Omron Sysmac Studio project modbus (Sysmac Studio 1.23.0.14, StandardProject)

# Controller new_Controller_0: NX1P2-1040DT1 version 1.18
Task PrimaryTask (priority 4, period or condition 2000): Programa0

VAR_GLOBAL CONSTANT
    Mi_Modulo485 : _sOPTBOARD_ID := (SlotNo := 2, IPAdr := [5(16#0)]);
END_VAR
VAR_GLOBAL
    Mi_Puerto : _sDEVICE_PORT;
    valor : INT;
    Escritura_20hz_Variador1 AT %W0.0 : BOOL;  (* published *)
    Escritura_50hz_Variador1 AT %W0.1 : BOOL;
END_VAR
VAR_GLOBAL RETAIN
    lectura_real AT %D0 : REAL;  (* published *)
END_VAR
VAR_GLOBAL
    run_fw : BOOL;
    run_bw : BOOL;
    stop_variador : BOOL;
    lectura_variador1 AT %W0.4 : BOOL;
    escritura_adelante_variador AT %W0.05 : BOOL;
    escritura_atras_variador AT %W0.06 : BOOL;
    escritura_marcha_variador AT %W0.2 : BOOL;
    escritura_paro_variador AT %W0.3 : BOOL;
    escritura_aceleracion1_variador : BOOL;
    escritura_aceleracion2_variador : BOOL;
END_VAR

PROGRAM Programa0
VAR
    Escritura_Frecuencia_Variador1 : BOOL;
    Instancia_Escritura_Frecuencia_Variador1 : NX_ModbusRtuWrite;
    Numero_Nodo_Variador1 : UINT;
    Trama_Escritura_Frecuencia_Variador1 : _sSERIAL_MODBUSRTU_WRITE;
    Datos_Escritura_Frecuencia_Variador1 : ARRAY[0..1] OF WORD;
    Option_Escritura_Frecuencia_Variador1 : _sSERIAL_MODBUSRTU_OPTION;
    Abort_Escritura_Frecuencia_Variador1 : BOOL;
    Busy_Escritura_Frecuencia_Variador1 : BOOL;
    CommandAborted_Escritura_Frecuencia_Variador1 : BOOL;
    Error_Escritura_Frecuencia_Variador1 : BOOL;
    ErrorID_Escritura_Frecuencia_Variador1 : BOOL;
    ErrorIDEX_Escritura_Frecuencia_Variador1 : BOOL;
    Instancia_Lectura_Frecuencia_Variador1 : NX_ModbusRtuRead;
    Trama_Lectura_Frecuencia_Variador1 : _sSERIAL_MODBUSRTU_READ;
    Datos_Lectura_Frecuencia_Variador1 : ARRAY[0..1] OF WORD;
    Option_Lectura_Frecuencia_Variador1 : _sSERIAL_MODBUSRTU_OPTION;
    Busy_Lectura_Frecuencia_Variador1 : BOOL;
    CommandAborted_Lectura_Frecuencia_Variador1 : BOOL;
    Error_Lectura_Frecuencia_Variador1 : BOOL;
    ErrorID_Lectura_Frecuencia_Variador1 : WORD;
    ErrorIDEX_Lectura_Frecuencia_Variador1 : DWORD;
    ReadSize_Lectura_Frecuencia_Variador1 : UINT;
    Abort_Lectura_Frecuencia_Variador1 : BOOL;
    nu : UINT;
    error : WORD;
    carmen : BOOL;
    pilo : BOOL;
    lectur : BOOL;
    Trama_Escritura_Marcha_Variador1 : _sSERIAL_MODBUSRTU_WRITE;
    Datos_Escritura_Marcha_Variador1 : BOOL;
    Option_Escritura_Marcha_Variador1 : _sSERIAL_MODBUSRTU_OPTION;
    Abort_Escritura_Marcha_Variador1 : BOOL;
    Trama_Escritura_Paro_Variador1 : _sSERIAL_MODBUSRTU_WRITE;
    Trama_Escritura_Sentido_Variador1 : _sSERIAL_MODBUSRTU_WRITE;
    Datos_Escritura_Sentido_Variador1 : BOOL;
    Option_Escritura_Sentido_Variador1 : _sSERIAL_MODBUSRTU_OPTION;
    Instancia_Escritura_Sentido_Variador1 : NX_ModbusRtuWrite;
    Datos_Escritura_Paro_Variador1 : BOOL;
    lectura_int : INT;
    Abort_Escritura_Sentido_Variador1 : BOOL;
    Trama_Escritura_Tiempo_Variador1 : _sSERIAL_MODBUSRTU_WRITE;
    Datos_Escritura_Tiempo_Variador1 : ARRAY[0..1] OF WORD;
    Option_Escritura_Tiempo_Variador1 : _sSERIAL_MODBUSRTU_OPTION;
    Abort_Escritura_Tiempo_Variador1 : BOOL;
END_VAR
VAR_EXTERNAL
    Mi_Puerto : _sDEVICE_PORT;
END_VAR
VAR_EXTERNAL CONSTANT
    Mi_Modulo485 : _sOPTBOARD_ID;
END_VAR
VAR_EXTERNAL
    Escritura_20hz_Variador1 : BOOL;
    Escritura_50hz_Variador1 : BOOL;
    lectura_variador1 : BOOL;
    escritura_adelante_variador : BOOL;
    escritura_atras_variador : BOOL;
    escritura_marcha_variador : BOOL;
    escritura_paro_variador : BOOL;
    lectura_real : REAL;
    escritura_aceleracion1_variador : BOOL;
    escritura_aceleracion2_variador : BOOL;
END_VAR

(* Section Escritura_Frecuencia_Variador1: ladder, written here as Structured Text *)

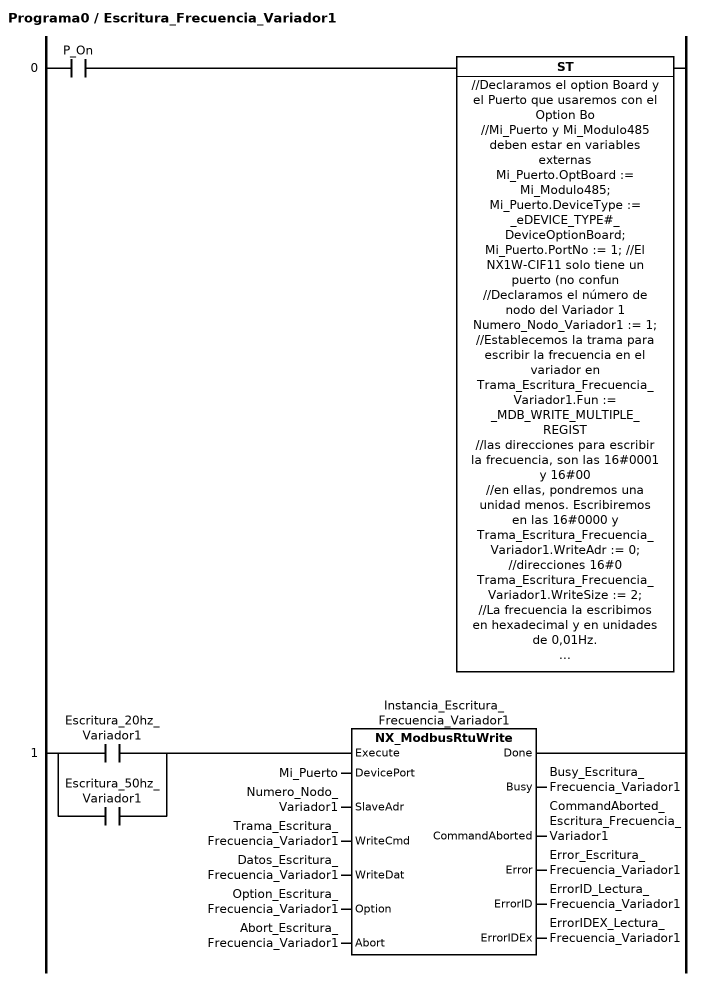
(* Rung 0 *)
IF P_On THEN
    //Declaramos el option Board y el Puerto que usaremos con el Option Board anterior.
    //Mi_Puerto y Mi_Modulo485 deben estar en variables externas
    Mi_Puerto.OptBoard := Mi_Modulo485;
    Mi_Puerto.DeviceType := _eDEVICE_TYPE#_DeviceOptionBoard;
    Mi_Puerto.PortNo := 1; //El NX1W-CIF11 solo tiene un puerto (no confundir con el slot donde está el módulo)
    
    //Declaramos el número de nodo del Variador 1
    Numero_Nodo_Variador1 := 1;
    
    //Establecemos la trama para escribir la frecuencia en el variador en los registros 0001h y 0002h
    Trama_Escritura_Frecuencia_Variador1.Fun := _MDB_WRITE_MULTIPLE_REGISTERS;
    //las direcciones para escribir la frecuencia, son las 16#0001 y 16#0002 pero como vamos a escribir
    //en ellas, pondremos una unidad menos. Escribiremos en las 16#0000 y 16#0001
    Trama_Escritura_Frecuencia_Variador1.WriteAdr := 0; //direcciones 16#0000 y 16#0001 para escribir la frecuencia
    Trama_Escritura_Frecuencia_Variador1.WriteSize := 2;
    
    //La frecuencia la escribimos en hexadecimal y en unidades de 0,01Hz. 5000 equivale a 50Hz.
    Datos_Escritura_Frecuencia_Variador1[0] := 0;
    IF Escritura_50hz_Variador1 THEN
    	Datos_Escritura_Frecuencia_Variador1[1] := 16#1388; //5000 en decimal que son 16#1388 (50Hz)
    ELSIF Escritura_20hz_Variador1 THEN
    	Datos_Escritura_Frecuencia_Variador1[1] := 16#07D0;
    END_IF;
    
    //establecemos que el TimeOut sea de 2 segundos (unidades de 0,1s) es el tiempo de espera
    //antes de dar por pérdida la comunicación y marcar el error 0400
    Option_Escritura_Frecuencia_Variador1.TimeOut := 20;
    
    //Activamos la comunicación poniendo la entrada Abort a False
    Abort_Escritura_Frecuencia_Variador1 := FALSE;
END_IF;
(* Rung 1 *)
Instancia_Escritura_Frecuencia_Variador1(Execute := Escritura_20hz_Variador1 OR Escritura_50hz_Variador1, DevicePort := Mi_Puerto, SlaveAdr := Numero_Nodo_Variador1, WriteCmd := Trama_Escritura_Frecuencia_Variador1, WriteDat := Datos_Escritura_Frecuencia_Variador1, Option := Option_Escritura_Frecuencia_Variador1, Abort := Abort_Escritura_Frecuencia_Variador1, Busy => Busy_Escritura_Frecuencia_Variador1, CommandAborted => CommandAborted_Escritura_Frecuencia_Variador1, Error => Error_Escritura_Frecuencia_Variador1, ErrorID => ErrorID_Lectura_Frecuencia_Variador1, ErrorIDEx => ErrorIDEX_Lectura_Frecuencia_Variador1);

(* Section Lectura_Frecuencia_Variador1: ladder, written here as Structured Text *)

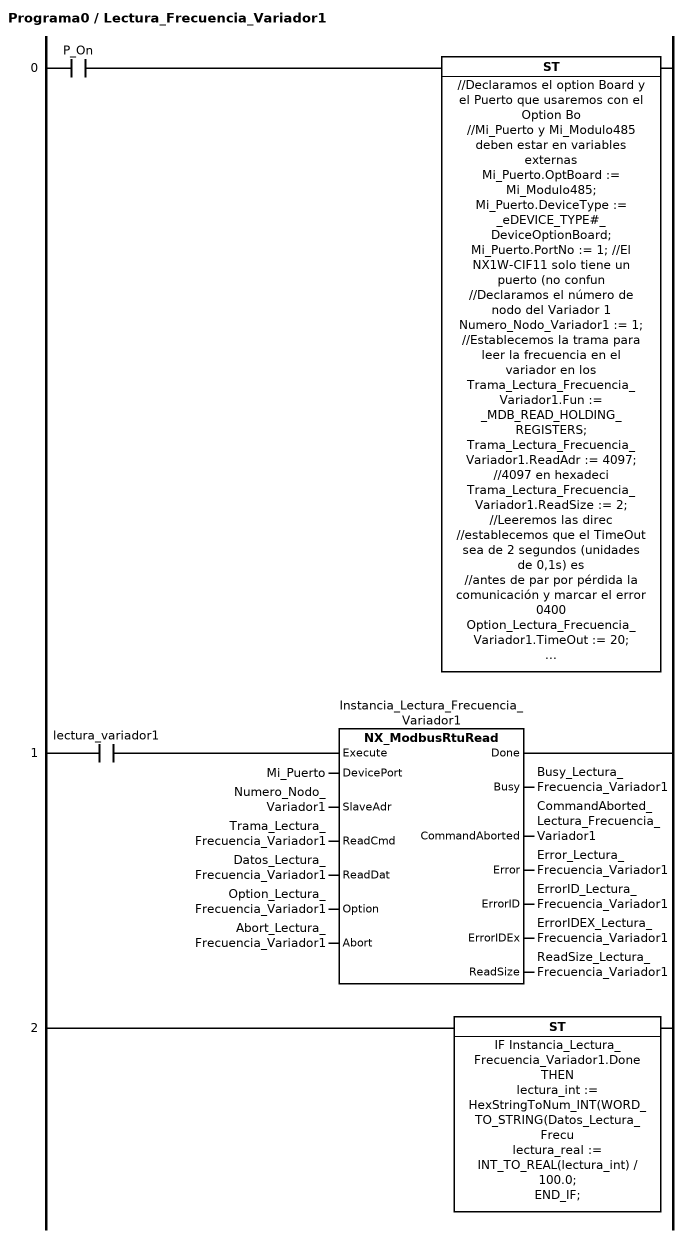
(* Rung 0 *)
IF P_On THEN
    //Declaramos el option Board y el Puerto que usaremos con el Option Board anterior.
    //Mi_Puerto y Mi_Modulo485 deben estar en variables externas
    Mi_Puerto.OptBoard := Mi_Modulo485;
    Mi_Puerto.DeviceType := _eDEVICE_TYPE#_DeviceOptionBoard;
    Mi_Puerto.PortNo := 1; //El NX1W-CIF11 solo tiene un puerto (no confundir con el slot donde está el módulo)
    
    //Declaramos el número de nodo del Variador 1
    Numero_Nodo_Variador1 := 1;
    
    //Establecemos la trama para leer la frecuencia en el variador en los registros 1001h y 1002h
    Trama_Lectura_Frecuencia_Variador1.Fun := _MDB_READ_HOLDING_REGISTERS;
    Trama_Lectura_Frecuencia_Variador1.ReadAdr := 4097; //4097 en hexadecimal es 16#1001
    Trama_Lectura_Frecuencia_Variador1.ReadSize := 2; //Leeremos las direcciones 16#1001 y 16#1002
    
    //establecemos que el TimeOut sea de 2 segundos (unidades de 0,1s) es el tiempo de espera
    //antes de par por pérdida la comunicación y marcar el error 0400
    Option_Lectura_Frecuencia_Variador1.TimeOut := 20;
    
    //Activamos la comunicación poniendo la entrada Abort a False
    Abort_Lectura_Frecuencia_Variador1 := FALSE;
END_IF;
(* Rung 1 *)
Instancia_Lectura_Frecuencia_Variador1(Execute := lectura_variador1, DevicePort := Mi_Puerto, SlaveAdr := Numero_Nodo_Variador1, ReadCmd := Trama_Lectura_Frecuencia_Variador1, ReadDat := Datos_Lectura_Frecuencia_Variador1, Option := Option_Lectura_Frecuencia_Variador1, Abort := Abort_Lectura_Frecuencia_Variador1, Busy => Busy_Lectura_Frecuencia_Variador1, CommandAborted => CommandAborted_Lectura_Frecuencia_Variador1, Error => Error_Lectura_Frecuencia_Variador1, ErrorID => ErrorID_Lectura_Frecuencia_Variador1, ErrorIDEx => ErrorIDEX_Lectura_Frecuencia_Variador1, ReadSize => ReadSize_Lectura_Frecuencia_Variador1);
(* Rung 2 *)
IF Instancia_Lectura_Frecuencia_Variador1.Done THEN
	lectura_int := HexStringToNum_INT(WORD_TO_STRING(Datos_Lectura_Frecuencia_Variador1[0]));
	lectura_real := INT_TO_REAL(lectura_int) / 100.0;
END_IF;

(* Section escritura_bit_marcha: ladder, written here as Structured Text *)

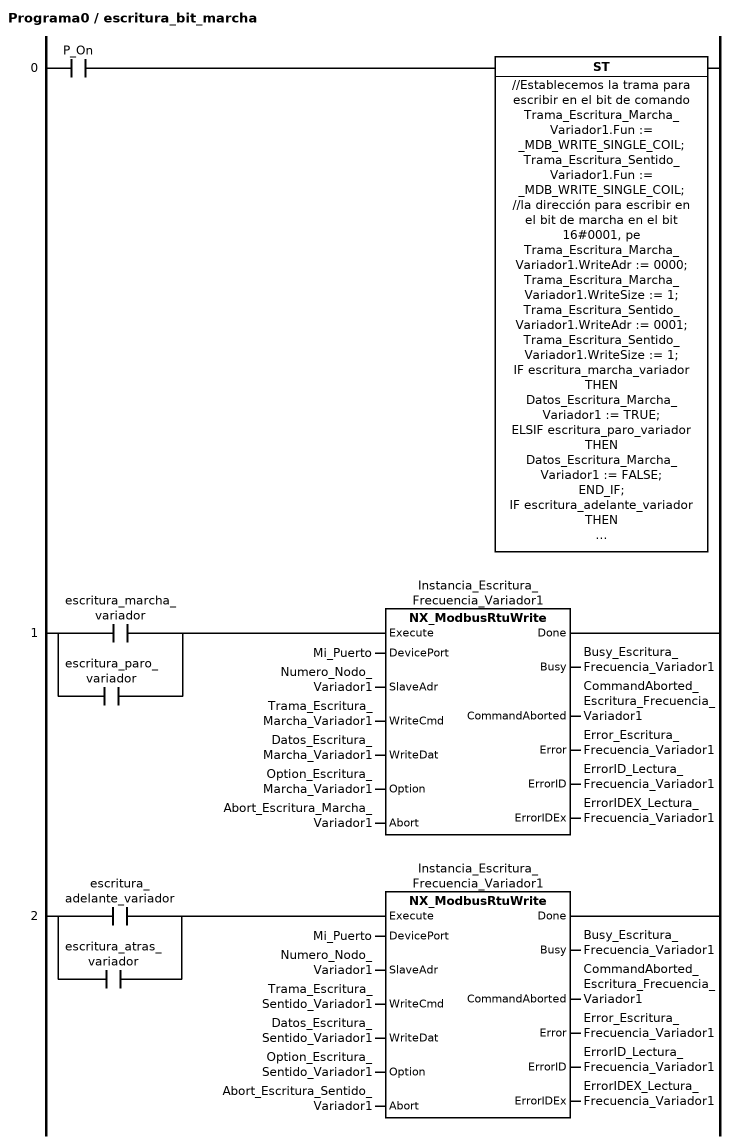
(* Rung 0 *)
IF P_On THEN
    //Establecemos la trama para escribir en el bit de comando
    Trama_Escritura_Marcha_Variador1.Fun := _MDB_WRITE_SINGLE_COIL;
    Trama_Escritura_Sentido_Variador1.Fun := _MDB_WRITE_SINGLE_COIL;
    //la dirección para escribir en el bit de marcha en el bit 16#0001, pero pondremos una unidad menos
    Trama_Escritura_Marcha_Variador1.WriteAdr := 0000;
    Trama_Escritura_Marcha_Variador1.WriteSize := 1;
    
    Trama_Escritura_Sentido_Variador1.WriteAdr := 0001;
    Trama_Escritura_Sentido_Variador1.WriteSize := 1;
    
    IF escritura_marcha_variador THEN
    	Datos_Escritura_Marcha_Variador1 := TRUE;
    ELSIF escritura_paro_variador THEN
    	Datos_Escritura_Marcha_Variador1 := FALSE;
    END_IF;
    
    IF escritura_adelante_variador THEN
    	Datos_Escritura_Sentido_Variador1 := TRUE;
    ELSIF escritura_atras_variador THEN
    	Datos_Escritura_Sentido_Variador1 := FALSE;
    END_IF;
    
    Option_Escritura_Marcha_Variador1.TimeOut := 20;
    Option_Escritura_Sentido_Variador1.TimeOut := 20;
    
    Abort_Escritura_Marcha_Variador1 := FALSE;
    Abort_Escritura_Sentido_Variador1 := FALSE;
END_IF;
(* Rung 1 *)
Instancia_Escritura_Frecuencia_Variador1(Execute := escritura_marcha_variador OR escritura_paro_variador, DevicePort := Mi_Puerto, SlaveAdr := Numero_Nodo_Variador1, WriteCmd := Trama_Escritura_Marcha_Variador1, WriteDat := Datos_Escritura_Marcha_Variador1, Option := Option_Escritura_Marcha_Variador1, Abort := Abort_Escritura_Marcha_Variador1, Busy => Busy_Escritura_Frecuencia_Variador1, CommandAborted => CommandAborted_Escritura_Frecuencia_Variador1, Error => Error_Escritura_Frecuencia_Variador1, ErrorID => ErrorID_Lectura_Frecuencia_Variador1, ErrorIDEx => ErrorIDEX_Lectura_Frecuencia_Variador1);
(* Rung 2 *)
Instancia_Escritura_Frecuencia_Variador1(Execute := escritura_adelante_variador OR escritura_atras_variador, DevicePort := Mi_Puerto, SlaveAdr := Numero_Nodo_Variador1, WriteCmd := Trama_Escritura_Sentido_Variador1, WriteDat := Datos_Escritura_Sentido_Variador1, Option := Option_Escritura_Sentido_Variador1, Abort := Abort_Escritura_Sentido_Variador1, Busy => Busy_Escritura_Frecuencia_Variador1, CommandAborted => CommandAborted_Escritura_Frecuencia_Variador1, Error => Error_Escritura_Frecuencia_Variador1, ErrorID => ErrorID_Lectura_Frecuencia_Variador1, ErrorIDEx => ErrorIDEX_Lectura_Frecuencia_Variador1);

(* Section sentido_marcha: ladder, written here as Structured Text *)

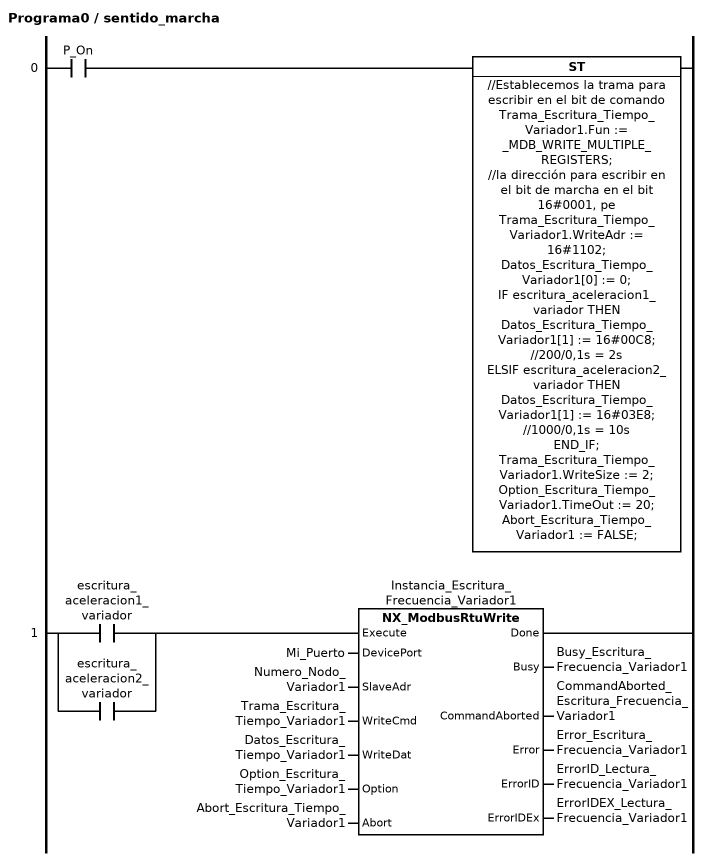
(* Rung 0 *)
IF P_On THEN
    //Establecemos la trama para escribir en el bit de comando
    Trama_Escritura_Tiempo_Variador1.Fun := _MDB_WRITE_MULTIPLE_REGISTERS;
    //la dirección para escribir en el bit de marcha en el bit 16#0001, pero pondremos una unidad menos
    Trama_Escritura_Tiempo_Variador1.WriteAdr := 16#1102;
    
    Datos_Escritura_Tiempo_Variador1[0] := 0;
    
    IF escritura_aceleracion1_variador THEN
    	Datos_Escritura_Tiempo_Variador1[1] := 16#00C8; //200/0,1s = 2s
    ELSIF escritura_aceleracion2_variador THEN
    	Datos_Escritura_Tiempo_Variador1[1] := 16#03E8; //1000/0,1s = 10s
    END_IF;
    
    Trama_Escritura_Tiempo_Variador1.WriteSize := 2;
    
    Option_Escritura_Tiempo_Variador1.TimeOut := 20;
    
    Abort_Escritura_Tiempo_Variador1 := FALSE;
END_IF;
(* Rung 1 *)
Instancia_Escritura_Frecuencia_Variador1(Execute := escritura_aceleracion1_variador OR escritura_aceleracion2_variador, DevicePort := Mi_Puerto, SlaveAdr := Numero_Nodo_Variador1, WriteCmd := Trama_Escritura_Tiempo_Variador1, WriteDat := Datos_Escritura_Tiempo_Variador1, Option := Option_Escritura_Tiempo_Variador1, Abort := Abort_Escritura_Tiempo_Variador1, Busy => Busy_Escritura_Frecuencia_Variador1, CommandAborted => CommandAborted_Escritura_Frecuencia_Variador1, Error => Error_Escritura_Frecuencia_Variador1, ErrorID => ErrorID_Lectura_Frecuencia_Variador1, ErrorIDEx => ErrorIDEX_Lectura_Frecuencia_Variador1);
END_PROGRAM

# Device HMI_NA5_0 (NA): not converted